FUNCTION_BLOCK AUDI_TO_AUDI2 (* Composite FB for convert unidirectional AUDI to bidirectional AUDI2 *)
  (* Standard: 61499-2; Function: AUDI_IN publishes its value onto the outgoing (EO1) side of AUDI2_BIDIR. Whatever AUDI2_BIDIR receives on its incoming (EI1) side is forwarded out again as a plain unidirectional signal via AUDI_OUT.; Description: Copyright (c) 2026 HR Agrartechnik GmbH This program and the accompanying materials are made available under the terms of the Eclipse Public License 2.0 which is available at https://www.eclipse.org/legal/epl-2.0/ SPDX-License-Identifier: EPL-2.0 *)
  (* Version 1.0, 2026-09-12, Franz Höpfinger, HR Agrartechnik GmbH, Initial Version - Konvertierungsfamilie vervollstaendigt (analog zu AR2/AB2/AE2). *)
  PACKAGE adapter::conversion::bidirectional;
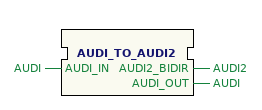
  SOCKETS
    AUDI_IN : adapter::types::unidirectional::AUDI; (* Adapter Input: unidirectional source *)
  END_SOCKETS
  PLUGS
    AUDI2_BIDIR : adapter::types::bidirectional::AUDI2; (* Adapter Output: bidirectional tap, outgoing side driven by AUDI_IN, incoming side forwarded to AUDI_OUT *)
    AUDI_OUT : adapter::types::unidirectional::AUDI; (* Adapter Output: mirrors AUDI2_BIDIR's incoming (request) side *)
  END_PLUGS
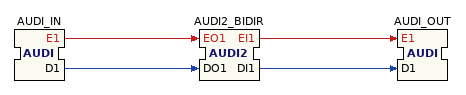
  EVENT_CONNECTIONS
    AUDI_IN.E1 TO AUDI2_BIDIR.EO1;
    AUDI2_BIDIR.EI1 TO AUDI_OUT.E1;
  END_CONNECTIONS
  DATA_CONNECTIONS
    AUDI_IN.D1 TO AUDI2_BIDIR.DO1;
    AUDI2_BIDIR.DI1 TO AUDI_OUT.D1;
  END_CONNECTIONS
END_FUNCTION_BLOCK
